INTERFACE I_Drive

{attribute 'monitoring':='call'}
PROPERTY Active : BOOL
GET
END_GET
END_PROPERTY

{attribute 'monitoring':='call'}
PROPERTY AtHome : BOOL
GET
END_GET
END_PROPERTY

{attribute 'monitoring':='call'}
PROPERTY Error : BOOL
GET
END_GET
END_PROPERTY

{attribute 'monitoring':='call'}
PROPERTY HomeSet : BOOL
GET
END_GET
END_PROPERTY

METHOD ABSTRACT homingSequence : BOOL
VAR_INPUT
END_VAR
END_METHOD

METHOD reset : BOOL
VAR_INPUT
END_VAR
END_METHOD

METHOD ABSTRACT stop : BOOL
VAR_INPUT
END_VAR
END_METHOD

METHOD toHome : BOOL
VAR_INPUT
END_VAR
END_METHOD

END_INTERFACE

(* stored: Version 1.1.0.1, ProductVersion 3.1.4024.11
   Itf I_Drive: Id {7acf7fde-0db8-42bf-8fcd-c1e82d306b2e}
   Property Active: Id {2682cd98-fc0a-42c6-9616-f63604b8ca6a}
   Get Get: Id {10e066ca-d04b-4480-a9db-66d31e276143}
   Property AtHome: Id {7daf1920-cf94-4627-a143-34e8d647584b}
   Get Get: Id {64157261-96dd-416a-9a58-3b0ce5cc71a5}
   Property Error: Id {c06dccc1-4c8f-42ec-9885-2ed6a0581fc4}
   Get Get: Id {3af5018b-1cfd-4805-a0ac-48e582a0aec0}
   Property HomeSet: Id {b41d4f54-374f-422d-ba91-2cb30a5412d2}
   Get Get: Id {0262e811-e4db-4230-b319-487b4f7ba9fd}
   Method homingSequence: Id {a9f91f05-b541-4dc6-a030-b69eac40ca8f}
   Method reset: Id {3bccf857-d910-47d2-bc88-8cbb1a53e9c0}
   Method stop: Id {a6446503-3ee0-4646-b748-8712ce55750a}
   Method toHome: Id {999a7a97-6c63-4f37-b0c0-03c4909e23c7} *)
